// TIA Portal project "Filling Water Tank With PLC and HMI" (V16)

(* hardware
DEVICE "S71500/ET200MP station_1"  S7-1500 station
   slot 0: "Rail_0"  Rack  6ES7 590-1***0-0AA0
   slot 1: "PLC_1"  CPU 1515-2 PN  6ES7 515-2AM01-0AB0  V2.8
      slot 3: "CPU display_1"  6ES7591-1BA00-0AA0
      slot 32768: "PROFINET interface_1"  X1
         slot 32769: "Port_1"  X1 P1
         slot 32770: "Port_2"  X1 P2
      slot 33024: "PROFINET interface_2"  X2
         slot 33025: "Port_1"  X2 P1
      slot 34817: "Virtual CP interface port_1"  Virtual CP interface port  Virtual CP interface port
DEVICE "HMI_1"  TP700 Comfort
   slot 0: "HMI_1"  TP700 Comfort  6AV2 124-0GC01-0AX0  16.0.0.0
   slot 1: "HMI_RT_1"  TP700 Comfort  6AV2 124-0GC01-0AX0  16.0.0.0
   slot 5: "HMI_1.IE_CP_1"  PROFINET Interface  16.0.0.0
      slot 1: "PROFINET Interface_1"  PROFINET Interface
         slot 1: "Port_1"  Port
         slot 2: "Port_2"  Port
   slot 7: "HMI_1.MPI/DP_CP_1"  MPI/DP Interface  16.0.0.0
*)

// ===== PLC "PLC_1"  CPU 1515-2 PN =====

VAR_GLOBAL   // PLC tag table "Default tag table"
   "Start PB" AT %M1.0 : Bool;
   "Cycle_On_mem_Bit" AT %M100.0 : Bool;
   "Stop PB" AT %M1.1 : Bool;
   "Low_LVL_Sens" AT %M1.3 : Bool;
   "Pump_1" AT %Q0.1 : Bool;
   "High_LVL_Sens" AT %M1.4 : Bool;
   "Pump_2" AT %Q0.2 : Bool;
   "Count" AT %MD50 : DWord;
   "Water_Tank_LVL" AT %MD54 : Real;
   "Tank_LVL_Mid" AT %M1.5 : Bool;
END_VAR

ORGANIZATION_BLOCK "Main"   // OB1, LAD, ProgramCycle
TITLE = "Main Program Sweep (Cycle)"
{ S7_Optimized_Access := 'TRUE' }
VERSION : 0.1
   VAR_INPUT
      Initial_Call : Bool;   // Initial call of this OB
      Remanence : Bool;   // =True, if remanent data are available
   END_VAR
   VAR_TEMP
      ret : Word;
   END_VAR
BEGIN

REGION Network 1
   // Start Stop Logic
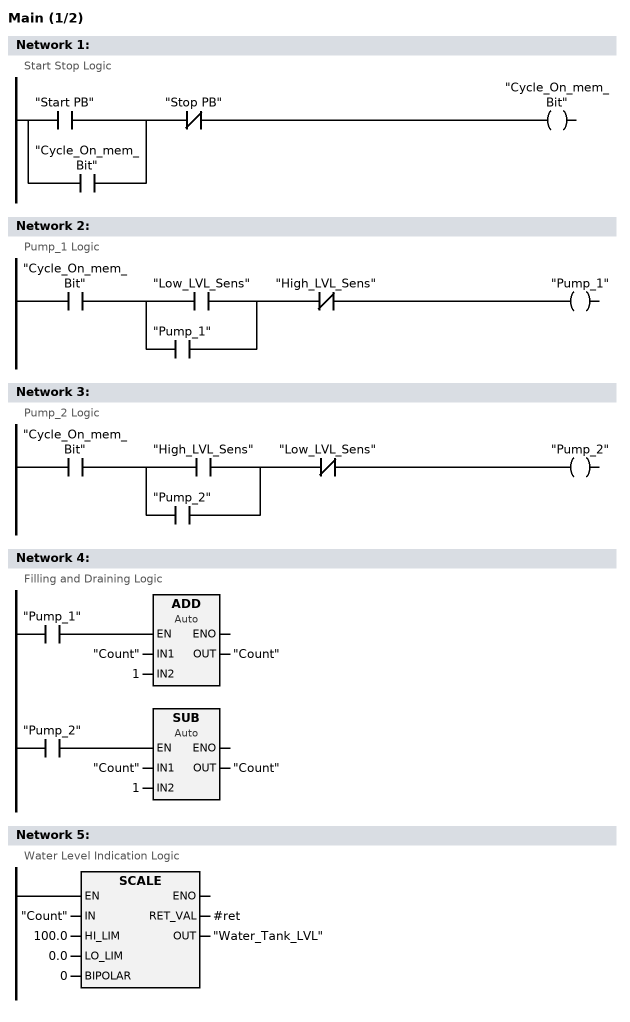
   RUNG wire#powerrail
      Contact( "Start PB" )
      wire#w1
      I_Contact( "Stop PB" )
      Coil( "Cycle_On_mem_Bit" )
   END_RUNG
   RUNG wire#powerrail
      Contact( "Cycle_On_mem_Bit" )
   END_RUNG wire#w1
   // the same network as SCL:
   "Cycle_On_mem_Bit" := ("Start PB" OR "Cycle_On_mem_Bit") AND NOT "Stop PB";
END_REGION

REGION Network 2
   // Pump_1 Logic
   RUNG wire#powerrail
      Contact( "Cycle_On_mem_Bit" )
      wire#w1
      Contact( "Low_LVL_Sens" )
      wire#w2
      I_Contact( "High_LVL_Sens" )
      Coil( "Pump_1" )
   END_RUNG
   RUNG wire#w1
      Contact( "Pump_1" )
   END_RUNG wire#w2
   // the same network as SCL:
   "Pump_1" := "Cycle_On_mem_Bit" AND ("Low_LVL_Sens" OR "Pump_1") AND NOT "High_LVL_Sens";
END_REGION

REGION Network 3
   // Pump_2 Logic
   RUNG wire#powerrail
      Contact( "Cycle_On_mem_Bit" )
      wire#w1
      Contact( "High_LVL_Sens" )
      wire#w2
      I_Contact( "Low_LVL_Sens" )
      Coil( "Pump_2" )
   END_RUNG
   RUNG wire#w1
      Contact( "Pump_2" )
   END_RUNG wire#w2
   // the same network as SCL:
   "Pump_2" := "Cycle_On_mem_Bit" AND ("High_LVL_Sens" OR "Pump_2") AND NOT "Low_LVL_Sens";
END_REGION

REGION Network 4
   // Filling and Draining Logic
   RUNG wire#powerrail
      Contact( "Pump_1" )
      Add(in1 := "Count", in2 := 1, out => "Count")
   END_RUNG
   RUNG wire#powerrail
      Contact( "Pump_2" )
      Sub(in1 := "Count", in2 := 1, out => "Count")
   END_RUNG
   // the same network as SCL:
   IF "Pump_1" THEN "Count" := "Count" + 1; END_IF;
   IF "Pump_2" THEN "Count" := "Count" - 1; END_IF;
END_REGION

REGION Network 5
   // Water Level Indication Logic
   #ret := SCALE(IN := "Count", HI_LIM := 100.0, LO_LIM := 0.0, BIPOLAR := 0, OUT => "Water_Tank_LVL");
END_REGION

REGION Network 6
   // Water Level Logic
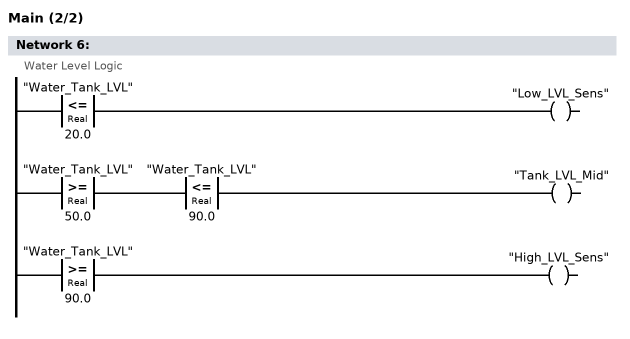
   RUNG wire#powerrail
      { S7_Templates := "SrcType := Real" } LE_Contact(in1 := "Water_Tank_LVL", in2 := 20.0)
      Coil( "Low_LVL_Sens" )
   END_RUNG
   RUNG wire#powerrail
      { S7_Templates := "SrcType := Real" } GE_Contact(in1 := "Water_Tank_LVL", in2 := 50.0)
      { S7_Templates := "SrcType := Real" } LE_Contact(in1 := "Water_Tank_LVL", in2 := 90.0)
      Coil( "Tank_LVL_Mid" )
   END_RUNG
   RUNG wire#powerrail
      { S7_Templates := "SrcType := Real" } GE_Contact(in1 := "Water_Tank_LVL", in2 := 90.0)
      Coil( "High_LVL_Sens" )
   END_RUNG
   // the same network as SCL:
   "Low_LVL_Sens" := "Water_Tank_LVL" <= 20.0;
   "Tank_LVL_Mid" := ("Water_Tank_LVL" >= 50.0) AND ("Water_Tank_LVL" <= 90.0);
   "High_LVL_Sens" := "Water_Tank_LVL" >= 90.0;
END_REGION
END_ORGANIZATION_BLOCK

(* ===== HMI "HMI_RT_1" =====
system functions are stored by id; their names below are inferred from use
connection "HMI_Connection_1": ETHERNET, S7_1500_OMS

HMI tags "Default tag table"
   "Tag_ScreenNumber" : UInt, internal
   "Start PB" : Bool = PLC "Start PB" AT %M1.0, 1 s
   "Stop PB" : Bool = PLC "Stop PB" AT %M1.1, 1 s
   "Low_LVL_Sens" : Bool = PLC Low_LVL_Sens AT %M1.3, 1 s
   "Tank_LVL_Mid" : Bool = PLC Tank_LVL_Mid AT %M1.5, 1 s
   "High_LVL_Sens" : Bool = PLC High_LVL_Sens AT %M1.4, 1 s
   "Water_Tank_LVL" : Real = PLC Water_Tank_LVL AT %MD54, 1 s
   "Pump_1" : Bool = PLC Pump_1 AT %Q0.1, 1 s
   "Pump_2" : Bool = PLC Pump_2 AT %Q0.2, 1 s

screen "Root screen" 800x420, template "Template_1"
   on GenerateScreen: SetTag("Tag_ScreenNumber", 1)
   Button "Button_1" at 48,23 size 96x32; TextOff 'Start'
      on Press: function_b14e0dd5("Start PB", 0)
      Appearance <- "Start PB"
   Button "Button_2" at 48,75 size 96x32; TextOff 'Stop'
      on Press: function_b14e0dd5("Stop PB", 0)
      Appearance <- "Stop PB"
   Bar "Bar_1" at 329,108 size 139x230; MinimumValue 0; MaximumValue 100
      ProcessValue <- "Water_Tank_LVL"
   SymbolLibrary "Symbol library_1" at 25,233 size 100x62
      Appearance <- "Pump_1"
   SymbolLibrary "Symbol library_2" at 319,54 size 44x55
   SymbolLibrary "Symbol library_3" at 121,250 size 120x24
   SymbolLibrary "Symbol library_4" at 240,227 size 54x47
   SymbolLibrary "Symbol library_5" at 267,107 size 27x121
   SymbolLibrary "Symbol library_6" at 267,54 size 53x54
   Button "Button_3" at 480,115 size 25x24; TextOff 'H'
      Appearance <- "High_LVL_Sens"
   Button "Button_4" at 481,191 size 26x24; TextOff 'M'
      Appearance <- "Tank_LVL_Mid"
   Button "Button_5" at 481,251 size 26x23; TextOff 'L'
      Appearance <- "Low_LVL_Sens"
   SymbolLibrary "Symbol library_7" at 541,289 size 67x61
      Appearance <- "Pump_2"
   SymbolLibrary "Symbol library_8" at 467,307 size 75x21
   SymbolLibrary "Symbol library_9" at 608,289 size 45x50
   TextField "Text field_1" at 544,221 size 113x23; Text 'Drain Motor'
   TextField "Text field_2" at 486,51 size 142x23; Text 'Level Indicator'
   TextField "Text field_3" at 23,180 size 120x23; Text 'Filling Motor'

Template "Template_1" 800x420
   Button "Exit" at 720,360 size 78x58; TextOff 'Exit'; PictureOff "ExitRuntime_TP700_Comfort_TR"; PictureOn "ExitRuntime_TP700_Comfort_TR"
      on Release: StopRuntime(0)
   Button "Template_Button" at 640,360 size 78x58; TextOff 'Text'
   Button "Template_Button_1" at 560,360 size 78x58; TextOff 'Text'
   Button "Template_Button_2" at 480,360 size 78x58; TextOff 'Text'
   Button "Template_Button_3" at 400,360 size 78x58; TextOff 'Text'
   Button "Template_Button_4" at 321,360 size 78x58; TextOff 'Text'
   Button "Template_Button_5" at 241,360 size 78x58; TextOff 'Text'
   Button "Template_Button_6" at 161,360 size 78x58; TextOff 'Text'
   Button "Alarms" at 81,360 size 78x58; TextOff 'Alarms'; PictureOff "AlarmDisplay_TP700_Comfort_TR"; PictureOn "AlarmDisplay_TP700_Comfort_TR"
      on Release: function_ef3f5d25("Alarm window_Unacknowledged", -1)
   Button "Start screen" at 1,360 size 78x58; TextOff 'Start screen'; PictureOff "NavigateHome_TP700_Comfort_TR"; PictureOn "NavigateHome_TP700_Comfort_TR"
      on Release: ActivateScreen("Root screen", 0)
*)